(*			
	EVERDE sp. z o.o.
	Rafał Osajda		22.01.2025		TC 4026.13		wer. 0.0.0.1
	B_Baza dla czujników binarnych 	
*)
FUNCTION_BLOCK INTERNAL ABSTRACT FB_Sensor EXTENDS FB_BaseComponent IMPLEMENTS ITF_Sensor, ITF_Sensor_HMI_Init
VAR
	bContact				AT %I*	: BOOL;		// Styk czujnika
	eType							: E_SensorType;
END_VAR

(*			
	EVERDE sp. z o.o.
	Rafał Osajda		05.02.2025		TC 4026.13		wer. 0.0.0.1
	Zwraca aktualny stan czujnika
*)
METHOD GetIsActive : BOOL
END_METHOD

METHOD PUBLIC GetSensorType : E_SensorType
VAR_INPUT
END_VAR
GetSensorType			:= THIS^.eType;
END_METHOD

METHOD PUBLIC GetSensorTypeToString : STRING
VAR CONSTANT
	arrType		: ARRAY [0..2] OF STRING := ['NO', 'NC', 'NOx2'];
END_VAR
GetSensorTypeToString			:= arrType [TO_INT (THIS^.eType)];
END_METHOD

END_FUNCTION_BLOCK

(* stored: Version 1.1.0.1
   POU FB_Sensor: Id {38d74651-ddd4-440f-81aa-c82978b08fa3}, SpecialFunc None
   Method GetIsActive: Id {db6dccc1-2a7a-463e-864e-da1a3729b042}
   Method GetSensorType: Id {f374bc07-fad7-40f2-bc55-235455285601}
   Method GetSensorTypeToString: Id {4ad723da-d327-4de9-9137-959624f49814} *)
